// TIA Portal V17 export
// export: Created 2022-10-18T15:35:35.600389Z, ExportSetting WithDefaults, DisplayName Totally Integrated Automation Portal, DisplayVersion V17 Update 5, DisplayName TIA Portal Openness, DisplayVersion V17 Update 5, DisplayName TIA Portal Teamcenter Gateway, DisplayVersion V17 Update 5, DisplayName TIA Portal Version Control Interface, DisplayVersion V17, DisplayName SINAMICS Startdrive Advanced, DisplayVersion V17 Update2, DisplayName SINAMICS Startdrive G130, G150, S120, S150, SINAMICS MV, S210, DisplayVersion V17 Update2, DisplayName SINAMICS Startdrive G110M, G120, G120C, G120D, G120P, G115D, DisplayVersion V17 Update2, DisplayName STEP 7 Professional, DisplayVersion V17 Update 5, DisplayName STEP 7 Safety, DisplayVersion V17, DisplayName WinCC Advanced / Unified PC, DisplayVersion V17 Update 5
FUNCTION "analogOutput" : Real   // FC2, LAD
{ S7_Optimized_Access := 'TRUE' }
VERSION : 0.1
// stored: AutoNumber true, IsIECCheckEnabled false, SetENOAutomatically false, UDAEnableTagReadback false
   VAR_INPUT
      setPoint : Real;
      minValueSensor : Real;
      maxValueSensor : Real;
   END_VAR
   VAR_OUTPUT
      scaledValue : Real;
   END_VAR
   VAR_TEMP
      normalizedValue : Real;
   END_VAR
   VAR CONSTANT
      MIN_VALUE : Int;
      MAX_VALUE : Int := 27648;
   END_VAR
BEGIN

REGION Network 1
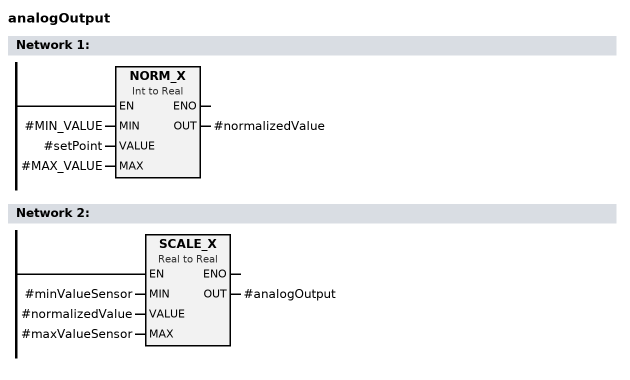
   RUNG wire#powerrail
      { S7_Templates := "[SrcType := Int, DestType := Real]" } Normalize(min := #MIN_VALUE, value := #setPoint, max := #MAX_VALUE, out => #normalizedValue)
   END_RUNG
   // the same network as SCL:
   #normalizedValue := NORM_X(MIN := #MIN_VALUE, VALUE := #setPoint, MAX := #MAX_VALUE);
END_REGION

REGION Network 2
   RUNG wire#powerrail
      { S7_Templates := "[SrcType := Real, DestType := Real]" } Scale(min := #minValueSensor, value := #normalizedValue, max := #maxValueSensor, out => #analogOutput)
   END_RUNG
   // the same network as SCL:
   #analogOutput := SCALE_X(MIN := #minValueSensor, VALUE := #normalizedValue, MAX := #maxValueSensor);
END_REGION
END_FUNCTION
